FUNCTION_BLOCK Attribute_IDA (* Input service interface function block for double word attribute input data *)
  (* Description: Copyright (c) 2017 fortiss GmbH, HR Agrartechnik GmbH This program and the accompanying materials are made available under the terms of the Eclipse Public License 2.0 which is available at https://www.eclipse.org/legal/epl-2.0/ SPDX-License-Identifier: EPL-2.0 *)
  (* Version 1.0, 2026-09-15, Franz Höpfinger, HR Agrartechnik GmbH, initial API and implementation and/or initial documentation *)
  PACKAGE isobus::UT::io::Attribute;
  IMPORT isobus::UT::Q::const::IDs::ID_NULL;
  IMPORT isobus::UT::io::Attribute::Attribute_ID;
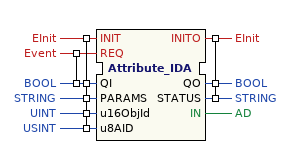
  EVENT_INPUT
    INIT : EInit WITH QI, PARAMS, u16ObjId, u8AID; (* Service Initialization *)
    REQ WITH QI; (* Service Request *)
  END_EVENT
  EVENT_OUTPUT
    INITO : EInit WITH QO, STATUS; (* Initialization Confirm *)
  END_EVENT
  VAR_INPUT
    QI : BOOL; (* Event Input Qualifier *)
    PARAMS : STRING; (* Service Parameters *)
    u16ObjId : UINT := ID_NULL; (* Object ID *)
    u8AID : USINT; (* Attribute ID of the object *)
  END_VAR
  VAR_OUTPUT
    QO : BOOL; (* Event Output Qualifier *)
    STATUS : STRING; (* Service Status *)
  END_VAR
  PLUGS
    IN : adapter::types::unidirectional::AD; (* Input data from resource *)
  END_PLUGS
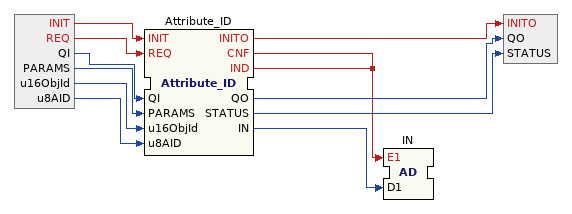
  FBS
    Attribute_ID : isobus::UT::io::Attribute::Attribute_ID;
  END_FBS
  EVENT_CONNECTIONS
    INIT TO Attribute_ID.INIT;
    REQ TO Attribute_ID.REQ;
    Attribute_ID.IND TO IN.E1;
    Attribute_ID.CNF TO IN.E1;
    Attribute_ID.INITO TO INITO;
  END_CONNECTIONS
  DATA_CONNECTIONS
    u16ObjId TO Attribute_ID.u16ObjId;
    u8AID TO Attribute_ID.u8AID;
    PARAMS TO Attribute_ID.PARAMS;
    QI TO Attribute_ID.QI;
    Attribute_ID.IN TO IN.D1;
    Attribute_ID.STATUS TO STATUS;
    Attribute_ID.QO TO QO;
  END_CONNECTIONS
END_FUNCTION_BLOCK
